(* CoDeSys 2.3.9.50 project: AdsClientTests.pro *)
(* Libraries: TcBase.lib 14.5.09 12:14:08, TcSystem.lib 7.6.16 11:01:22, TcSystemCX.lib 7.9.16 12:51:26, STANDARD.LIB 5.6.98 12:03:02, TcDataExchange.lib 10.8.16 15:23:34 *)

(* Task configuration *)
TASK Standard (PRIORITY := 0, INTERVAL := T#10ms);
	PRG_AdsClientTests
END_TASK

(* Global variable list: AdsClientTests/GVL_AdsClientTests *)
VAR_GLOBAL
	VERSION	: STRING := '2.0.0';
	IsReset 		: BOOL := TRUE;
	IsTestProject 	: BOOL := TRUE;
	IsRunning 	: BOOL;
	TestPointer 	: POINTER TO BOOL; (*//FOR 32/64bit check*)
	IsTc2 		: BOOL := TRUE;
END_VAR

(* Global variable list: AdsClientTests/GVL_Read *)
VAR_GLOBAL
	StandardTypes 		: ST_StandardTypes;
	StandardArrays 		: ST_StandardArrayTypes;
	ComplexTypes		: ST_ComplexTypes;
	ComplexArrayTypes	: ST_ComplexArrayTypes;
	SpecialTypes		: ST_SpecialTypes;
	IssueSpecificTypes	: ST_IssueSpecificTypes;
END_VAR

(* Global variable list: AdsClientTests/GVL_Subscription *)
VAR_GLOBAL
	NumericValue_10ms		 : INT;
	NumericValue_100ms 		: INT;
	NumericValue_1000ms 	: INT;
	Numericvalue_Constant	: INT := 12245;
END_VAR

(* Global variable list: AdsClientTests/GVL_SymbolsAndDataTypes *)
VAR_GLOBAL PERSISTENT
	TestSymbol : STRING(82) := 'Some test value';(*Test comment äääöö*)
	TestDataType : ST_TestDataType;
END_VAR

(* Global variable list: AdsClientTests/GVL_Write *)
VAR_GLOBAL
	Write_StandardTypes 		: ST_StandardTypes;
	Write_StandardArrays 		: ST_StandardArrayTypes;
	Write_ComplexTypes		: ST_ComplexTypes;
	Write_ComplexArrayTypes	: ST_ComplexArrayTypes;
	Write_SpecialTypes		: ST_SpecialTypes;
	Write_IssueSpecificTypes	: ST_IssueSpecificTypes;
END_VAR

(* Data type *)
TYPE E_Enum :
(
	Disabled 	:= 0,
	Starting 		:= 50,
	Running 		:= 100,
	Stopping		:= 200,
	Unknown		:= -99
);
END_TYPE

(* Data type *)
TYPE ST_ComplexArrayTypes :
STRUCT
	STRUCT_ 	: ARRAY[0..2] OF ST_StandardTypes;
	STRUCT_2 	: ARRAY[0..2] OF ST_StandardArrayTypes;
	ALIAS_ 		: ARRAY[0..2] OF StandardTypesAlias;
	ENUM_		: ARRAY[0..2] OF E_Enum := Running, Disabled, Stopping;
	ENUM_2		: ARRAY[0..2] OF E_Enum := Unknown, Disabled, Starting;
	ENUM_3		: ARRAY[0..2] OF E_Enum :=5555, 0, Unknown;
	POINTER_	: ARRAY[0..2] OF POINTER TO ST_StandardTypes;
	SUBRANGE_	: ARRAY[0..2] OF INT(-4095..4095) := 1234, 0, -1234;
	BLOCK_		: ARRAY[0..2] OF FB_Block :=
		(StrValue := 'First'),
		(StrValue := ''),
		(StrValue := 'Third')
	;
	BLOCK_2		: ARRAY[0..2] OF TON := (PT := T#2S500MS), (), (PT := T#123S);
	BLOCK_3		: ARRAY[0..2] OF FB_CreateDir :=
		(sPathName := 'C:\Test'),
		(),
		(sPathName := 'C:\AnotherTest')
	;
	BLOCK_4		: ARRAY[0..2] OF FB_ReadAdsSymByName :=
		(sVarName := 'GVL_Test.Variable'),
		(),
		(sVarName := 'GVL_Test.AnotherVariable')
	;
END_STRUCT
END_TYPE

(* Data type *)
TYPE ST_ComplexTypes :
STRUCT
	STRUCT_ 	: ST_StandardTypes;
	STRUCT_2 	: ST_StandardArrayTypes;
	ALIAS_ 		: StandardTypesAlias;
	ENUM_		: E_Enum := Running;
	ENUM_2		: E_Enum := Unknown;
	ENUM_3		: E_Enum := 5555; (*//Not a valid value*)
	POINTER_	: POINTER TO ST_StandardTypes;
	SUBRANGE_	: INT(-4095..4095) := 1234;
	BLOCK_		: FB_Block;
	BLOCK_2	: TON := (PT := T#2S500MS);
	BLOCK_3	: FB_CreateDir := (sPathName := 'C:\Test');
	BLOCK_4	: FB_ReadAdsSymByName := (sVarName := 'GVL_Test.Variable');
END_STRUCT
END_TYPE

(* Data type *)
TYPE ST_Issue94 :
STRUCT
	BoolValue 	: BOOL := TRUE;
	ArrayValue 	:  ARRAY [0..1] OF ST_Issue94_Byte := (ByteValue := 1), (ByteValue := 2);
END_STRUCT
END_TYPE

(* Data type *)
TYPE ST_Issue94_Byte :
STRUCT
	ByteValue : BYTE;
END_STRUCT
END_TYPE

(* Data type *)
TYPE ST_IssueSpecificTypes :
STRUCT
	Issue94	: ST_Issue94;
END_STRUCT
END_TYPE

(* Data type *)
TYPE ST_SpecialTypes :
STRUCT
	NegativeIndexArray		: ARRAY[-100..100] OF LREAL := 1.11, 99(0.0), 5.55, 99(0.0), 9.99;
	MultiDimensionalArray		: ARRAY[1..3, 1..2] OF BYTE := 1, 2, 3, 4, 5, 6;
	ArrayOfArrays			: ARRAY[1..3] OF ARRAY[1..2] OF SINT :=-1, -2, -3, -4, -5, -6;

	EmptyBlock		: FB_EmptyBlock;
	EmptyArray 		: ARRAY[0..-1] OF BOOL; (*How is this even possible..?*)
END_STRUCT
END_TYPE

(* Data type *)
TYPE ST_StandardArrayTypes :
STRUCT
	BOOL_ 	: ARRAY[0..2] OF BOOL := TRUE, FALSE, TRUE;
	BOOL_2 	: ARRAY[0..2] OF BOOL := FALSE, TRUE, FALSE;
	BYTE_ 	: ARRAY[0..2] OF BYTE := 255, 254, 0;
	WORD_ 	: ARRAY[0..2] OF WORD := 65535, 65534, 0;
	DWORD_ 	: ARRAY[0..2] OF DWORD := 4294967295, 4294967294, 0;
	SINT_ 	: ARRAY[0..2] OF SINT := 127, 126, 0;
	SINT_2 	: ARRAY[0..2] OF SINT := -128, -127, 0;
	USINT_ 	: ARRAY[0..2] OF USINT := 255, 254, 0;
	INT_ 	: ARRAY[0..2] OF INT := 32767, 0, -32768;
	INT_2 	: ARRAY[0..2] OF INT := -32768, 0, 32767;
	UINT_ 	: ARRAY[0..2] OF UINT := 65535, 65534, 0;
	DINT_ 	: ARRAY[0..2] OF DINT := 2147483647, 0, -2147483648;
	DINT_2 	: ARRAY[0..2] OF DINT := -2147483648, 0, 2147483647;
	UDINT_ 	: ARRAY[0..2] OF UDINT := 4294967295, 4294967294, 0;
	REAL_ 	: ARRAY[0..2] OF REAL := 3.4E38, 0, -3.4E38;
	REAL_2 	: ARRAY[0..2] OF REAL := -3.4E38, 0, 3.4E38;
	REAL_3 	: ARRAY[0..2] OF REAL := 75483.545, 0, -75483.545;
	REAL_4 	: ARRAY[0..2] OF REAL := -75483.545, 0, 75483.545;
	STRING_	: ARRAY[0..2] OF STRING := 'A test string ääöö!!@@', '', 'String value';
	STRING_2: ARRAY[0..2] OF STRING(255) :=
		'Lorem ipsum dolor sit amet, consectetur adipiscing elit. Pellentesque bibendum mauris vel metus rutrum, sed gravida justo dignissim. Aenean et nisi cursus, auctor mi vel, posuere enim. Suspendisse ultricies mauris in finibus tristique. Nullam turpis duis.',
		'',
		'Proin tempor diam a felis fermentum, id molestie tortor pharetra. Phasellus condimentum rhoncus ultrices. Suspendisse ultricies nec neque quis sodales. In molestie vestibulum nulla eu gravida. Morbi orci ipsum, gravida elementum eros non, egestas egestas.';
	DATE_ 	: ARRAY[0..2] OF DATE := D#2106-02-06, D#2106-02-05;
	DT_ 	: ARRAY[0..2] OF DT := DT#2106-02-06-06:28:15, DT#2106-02-06-06:28:14;
	DT_2 	: ARRAY[0..2] OF DATE_AND_TIME := DT#2106-02-06-06:28:15, DT#2106-02-06-06:28:14;
	TOD_ 	: ARRAY[0..2] OF TOD;
	TOD_2 	: ARRAY[0..2] OF TIME_OF_DAY;
	TIME_ 	: ARRAY[0..2] OF TIME := T#49D17H2M47S295MS, T#49D17H2M47S294MS, T#0S;
	LREAL_ 	: ARRAY[0..2] OF LREAL := 1.7E308, 0, -1.7E308;
	LREAL_2 : ARRAY[0..2] OF LREAL := -1.7E308, 0, 1.7E308;
	LREAL_3	: ARRAY[0..2] OF REAL := 75483.545, 0, -75483.545;
	LREAL_4	: ARRAY[0..2] OF REAL := -75483.545, 0, 75483.545;
END_STRUCT
END_TYPE

(* Data type *)
TYPE ST_StandardTypes :
STRUCT
	BOOL_ 	: BOOL := TRUE;
	BOOL_2 	: BOOL := FALSE;
	BYTE_ 	: BYTE := 255;
	WORD_ 	: WORD := 65535;
	DWORD_ 	: DWORD := 4294967295;
	SINT_ 	: SINT := 127;
	SINT_2 	: SINT := -128;
	USINT_ 	: USINT := 255;
	INT_ 	: INT := 32767;
	INT_2 	: INT := -32768;
	UINT_ 	: UINT := 65535;
	DINT_ 	: DINT := 2147483647;
	DINT_2 	: DINT := -2147483648;
	UDINT_ 	: UDINT := 4294967295;
	REAL_ 	: REAL := 3.4E38;
	REAL_2 	: REAL := -3.4E38;
	REAL_3 	: REAL := 75483.545;
	REAL_4 	: REAL := -75483.545;
	STRING_	: STRING := 'A test string ääöö!!@@';
	STRING_2: STRING(255) := 'Lorem ipsum dolor sit amet, consectetur adipiscing elit. Pellentesque bibendum mauris vel metus rutrum, sed gravida justo dignissim. Aenean et nisi cursus, auctor mi vel, posuere enim. Suspendisse ultricies mauris in finibus tristique. Nullam turpis duis.';
	DATE_ 	: DATE := D#2106-02-06;
	DT_ 	: DT := DT#2106-02-06-06:28:15;
	DT_2 	: DATE_AND_TIME := DT#2106-02-06-06:28:15;
	TOD_ 	: TOD;
	TOD_2 	: TIME_OF_DAY;
	TIME_ 	: TIME := T#49D17H2M47S295MS;
	LREAL_ 	: LREAL := 1.7E308;
	LREAL_2 : LREAL := -1.7E308;
	LREAL_3 : REAL := 75483.545;
	LREAL_4 : REAL := -75483.545;
END_STRUCT
END_TYPE

(* Data type *)
TYPE ST_Struct :
STRUCT
	SomeText : STRING(50) := 'Hello ads-client';
	SomeReal : REAL := 3.14159265359;
	SomeDate : DT := DT#2020-4-13-12:25:33;
END_STRUCT
END_TYPE

(* Data type *)
(*Test comment äääöö*)
TYPE ST_TestDataType :
STRUCT
	Member : ST_Struct;
END_STRUCT
END_TYPE

(* Data type *)
TYPE StandardTypesAlias : ST_StandardTypes; END_TYPE

(* POU PRG_AdsClientTests, ST *)
PROGRAM PRG_AdsClientTests
VAR
	InitDone : BOOL;

	TOD_0: TOD;
	TOD_MAX : TOD;
	TOD_MAX_MINUS_1 : TOD;
END_VAR
IF NOT IsRunning THEN
	(*Need to do some initializing here unlike in TC3*)
	TOD_0 := DWORD_TO_TOD(0);
	TOD_MAX := DWORD_TO_TOD(4294967295);
	TOD_MAX_MINUS_1 := DWORD_TO_TOD(4294967294);

	StandardArrays.TOD_[0] := TOD_MAX;
	StandardArrays.TOD_[1] := TOD_MAX_MINUS_1;
	StandardArrays.TOD_[2] := TOD_0;
	StandardArrays.TOD_2[0] := TOD_MAX;
	StandardArrays.TOD_2[1] := TOD_MAX_MINUS_1;
	StandardArrays.TOD_2[2] := TOD_0;

	StandardTypes.TOD_ := TOD_MAX;
	StandardTypes.TOD_2 := TOD_MAX;

	ComplexTypes.POINTER_ := ADR(StandardTypes);

	ComplexTypes.BLOCK_.Data.TOD_  := TOD_MAX;
	ComplexTypes.BLOCK_.Data.TOD_2  := ComplexTypes.BLOCK_.Data.TOD_;

	ComplexTypes.ALIAS_.TOD_  := ComplexTypes.BLOCK_.Data.TOD_;
	ComplexTypes.ALIAS_.TOD_2  := ComplexTypes.BLOCK_.Data.TOD_;

	ComplexTypes.STRUCT_.TOD_  := ComplexTypes.BLOCK_.Data.TOD_;
	ComplexTypes.STRUCT_.TOD_2  := ComplexTypes.BLOCK_.Data.TOD_;

	ComplexTypes.STRUCT_2.TOD_[0]  := TOD_MAX;
	ComplexTypes.STRUCT_2.TOD_[1]  := TOD_MAX_MINUS_1;
	ComplexTypes.STRUCT_2.TOD_[2]  := TOD_0;
	ComplexTypes.STRUCT_2.TOD_2[0]  := TOD_MAX;
	ComplexTypes.STRUCT_2.TOD_2[1]  := TOD_MAX_MINUS_1;
	ComplexTypes.STRUCT_2.TOD_2[2]  := TOD_0;

	ComplexArrayTypes.BLOCK_[0].Data.TOD_  := TOD_MAX;
	ComplexArrayTypes.BLOCK_[0].Data.TOD_2  := TOD_MAX;
	ComplexArrayTypes.BLOCK_[1].Data.TOD_  := TOD_MAX;
	ComplexArrayTypes.BLOCK_[1].Data.TOD_2  := TOD_MAX;
	ComplexArrayTypes.BLOCK_[2].Data.TOD_  := TOD_MAX;
	ComplexArrayTypes.BLOCK_[2].Data.TOD_2  := TOD_MAX;

	ComplexArrayTypes.ALIAS_[0].TOD_  := TOD_MAX;
	ComplexArrayTypes.ALIAS_[0].TOD_2  := TOD_MAX;
	ComplexArrayTypes.ALIAS_[1].TOD_  := TOD_MAX;
	ComplexArrayTypes.ALIAS_[1].TOD_2  := TOD_MAX;
	ComplexArrayTypes.ALIAS_[2].TOD_  := TOD_MAX;
	ComplexArrayTypes.ALIAS_[2].TOD_2  := TOD_MAX;

	ComplexArrayTypes.STRUCT_[0].TOD_  := TOD_MAX;
	ComplexArrayTypes.STRUCT_[0].TOD_2  := TOD_MAX;
	ComplexArrayTypes.STRUCT_[1].TOD_  := TOD_MAX;
	ComplexArrayTypes.STRUCT_[1].TOD_2  := TOD_MAX;
	ComplexArrayTypes.STRUCT_[2].TOD_  := TOD_MAX;
	ComplexArrayTypes.STRUCT_[2].TOD_2  := TOD_MAX;

	ComplexArrayTypes.STRUCT_2[0].TOD_[0]  := TOD_MAX;
	ComplexArrayTypes.STRUCT_2[0].TOD_[1]  := TOD_MAX_MINUS_1;
	ComplexArrayTypes.STRUCT_2[0].TOD_[2]  := TOD_0;
	ComplexArrayTypes.STRUCT_2[0].TOD_2[0]  := TOD_MAX;
	ComplexArrayTypes.STRUCT_2[0].TOD_2[1]  := TOD_MAX_MINUS_1;
	ComplexArrayTypes.STRUCT_2[0].TOD_2[2]  := TOD_0;

	ComplexArrayTypes.STRUCT_2[1] := ComplexArrayTypes.STRUCT_2[0];
	ComplexArrayTypes.STRUCT_2[2] := ComplexArrayTypes.STRUCT_2[0];

	MEMSET(ADR(Write_StandardTypes), 0, SIZEOF(Write_StandardTypes));
	MEMSET(ADR(Write_StandardTypes), 0, SIZEOF(Write_StandardArrays));
	MEMSET(ADR(Write_ComplexTypes), 0, SIZEOF(Write_ComplexTypes));
	MEMSET(ADR(Write_ComplexArrayTypes), 0, SIZEOF(Write_ComplexArrayTypes));
	MEMSET(ADR(Write_SpecialTypes), 0, SIZEOF(Write_SpecialTypes));
	MEMSET(ADR(Write_IssueSpecificTypes), 0, SIZEOF(Write_IssueSpecificTypes));

	Write_ComplexTypes.POINTER_ := ADR(Write_StandardTypes);
	
	IsRunning := TRUE;
END_IF

PRG_Subscription();
END_PROGRAM

(* POU PRG_Subscription, ST *)
PROGRAM PRG_Subscription
VAR
	tonUpdate10ms : ton;
	tonUpdate100ms : ton;
	tonUpdate1000ms : TON;
END_VAR
(*//-------------------
// 10 ms
//-------------------*)
tonUpdate10ms(
	IN := TRUE,
	PT := T#10MS
);

IF tonUpdate10ms.Q THEN
	NumericValue_10ms := NumericValue_10ms + 1;

	tonUpdate10ms(IN := FALSE);
	tonUpdate10ms(IN := TRUE);
END_IF

(*//-------------------
// 100 ms
//-------------------*)
tonUpdate100ms(
	IN := TRUE,
	PT := T#100MS
);

IF tonUpdate100ms.Q THEN
	NumericValue_100ms := NumericValue_100ms + 1;

	tonUpdate100ms(IN := FALSE);
	tonUpdate100ms(IN := TRUE);
END_IF

(*//-------------------
// 1000 ms
//-------------------*)
tonUpdate1000ms(
	IN := TRUE,
	PT := T#1000MS
);

IF tonUpdate1000ms.Q THEN
	NumericValue_1000ms := NumericValue_1000ms + 1;

	tonUpdate1000ms(IN := FALSE);
	tonUpdate1000ms(IN := TRUE);
END_IF
END_PROGRAM

(* POU FB_Block, ST *)
(*Variables in inputs so that they can be written from outside*)
FUNCTION_BLOCK FB_Block
VAR_INPUT
	StrValue : STRING;
	Data : ST_StandardTypes;
END_VAR
VAR_OUTPUT
END_VAR
VAR
END_VAR
;
END_FUNCTION_BLOCK

(* POU FB_EmptyBlock, ST *)
FUNCTION_BLOCK FB_EmptyBlock
VAR_INPUT
END_VAR
VAR_OUTPUT
END_VAR
VAR
END_VAR
;
END_FUNCTION_BLOCK
